FUNCTION_BLOCK FB_ActorRotateCCWCommand IMPLEMENTS I_Command
VAR
	refFlyingHoist : REFERENCE TO FB_FlyingHoist;
END_VAR

METHOD Execute
IF (__ISVALIDREF(THIS^.refFlyingHoist)) THEN
	THIS^.refFlyingHoist.HoistEnable();
	THIS^.refFlyingHoist.ActorRotateCCW();
END_IF
END_METHOD

METHOD FB_init : BOOL
VAR_INPUT
	bInitRetains 	: BOOL; // if TRUE, the retain variables are initialized (warm start / cold start)
	bInCopyCode 	: BOOL;  // if TRUE, the instance afterwards gets moved into the copy code (online change)
	refFlyingHoist 	: REFERENCE TO FB_FlyingHoist;
END_VAR
IF (__ISVALIDREF(refFlyingHoist)) THEN
	THIS^.refFlyingHoist REF= refFlyingHoist;
ELSE
	THIS^.refFlyingHoist REF= 0;
END_IF
END_METHOD

END_FUNCTION_BLOCK

(* stored: Version 1.1.0.1, ProductVersion 3.1.4022.18
   POU FB_ActorRotateCCWCommand: Id {741dd56c-c740-439b-a04b-43b7462a92eb}, SpecialFunc None
   Method Execute: Id {4984f520-6602-49c5-bfe2-d6a0337076d4}
   Method FB_init: Id {c6449c30-ae6f-419c-8bf6-b698a64e097f} *)
